FUNCTION F_Messages : BOOL
VAR_INPUT
END_VAR
VAR
END_VAR

;
{text'hello world'}
{info'information'}
{warn'warning'}
//{error'Error!'}

END_FUNCTION

(* stored: Version 1.1.0.1, ProductVersion 3.1.4024.2
   POU F_Messages: Id {ff8464c9-d904-4617-be35-eb0c8e685418}, SpecialFunc None *)
